PROGRAM FB_ExportCSV
VAR_INPUT
	bExport				: BOOL;
END_VAR

VAR
	hr : HRESULT;
	
	fbCsvExportSetting	: FB_TcEventCsvExportSettings; 
	fbExportFilter		: I_TcEventFilter; 
	sExportFilePath		: T_maxString := 'C:\dataCollection\';
	sExportFileName		: T_maxString := 'Alarms_History.csv';
	
	fbEventLogger	: FB_TcEventLogger;
	fbTrig			: R_TRIG;
	
	getTime : FB_LocalSystemTime := ( bEnable := TRUE, dwCycle := 5 );
	dateStr : T_MaxString;
END_VAR

getTime();
fbTrig(CLK:=bExport);
IF bExport THEN
	IF fbTrig.Q THEN 
		dateStr := getDateStr();
		sExportFileName	:= Concat(Concat(sExportFilePath,'Alarms_History_'),Concat(dateStr,'.csv'));
		fbCsvExportSetting.Clear();
		fbCsvExportSetting.sDelimiter := ',' ;
		//fbCsvExportSetting.AddLanguage(1031, 'German');
		fbCsvExportSetting.AddFilter(fbExportFilter); 
		//fbExportFilter.Clear().IsMessage().AND_OP().EventClass.EqualTo(TC_EVENTS.Alarm.Event.uuidEventClass);
	END_IF
	IF fbEventLogger.ExportLoggedEvents(sExportFileName, fbCsvExportSetting, hrErrorCode=>hr) THEN // async request returns TRUE if not any more busy 
		bExport := FALSE;
	END_IF
END_IF

METHOD getDateStr : T_MaxString
VAR_INPUT
END_VAR
getDateStr := CONCAT(WORD_TO_STRING(getTime.systemTime.wMonth), CONCAT('_', CONCAT(WORD_TO_STRING(getTime.systemTime.wDay), CONCAT('_', WORD_TO_STRING(getTime.systemTime.wYear)))));
END_METHOD

END_PROGRAM

(* stored: Version 1.1.0.1, ProductVersion 3.1.4024.6
   POU FB_ExportCSV: Id {2803cd03-f8cf-4705-b3e1-f7317ef61984}, SpecialFunc None
   Method getDateStr: Id {e57e5c5d-98ed-499d-a978-808d7703ecac} *)
